(* CODESYS project Screen_1.xml

Project tree, tasks and I/O mapping:
  visualisation Screen_1
*)

// /Screen_1
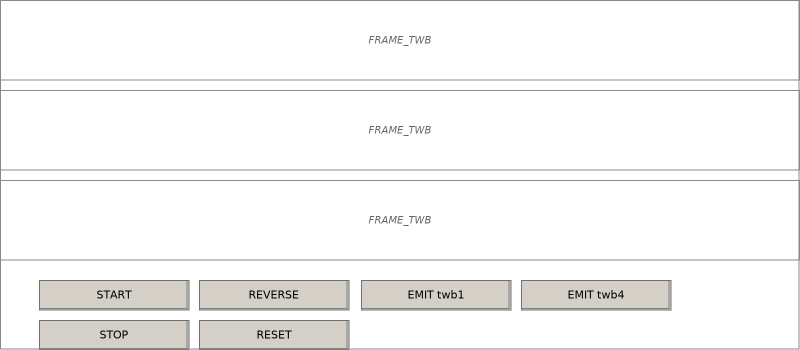
VISUALIZATION Screen_1  // 800x350
    Frame (0,0 800x80)
        shows FRAME_TWB(conveyor := ZONE_HMI.arConveyors[1])
    Frame (0,90 800x80)
        shows FRAME_TWB(conveyor := ZONE_HMI.arConveyors[2])
    Frame (0,180 800x80)
        shows FRAME_TWB(conveyor := ZONE_HMI.arConveyors[3])
    Button (39,280 150x30), "START"
        OnMouseClick: execute { ZONE_HMI.xStart := TRUE; }
    Button (199,280 150x30), "REVERSE"
        OnMouseClick:  ToggleVariable=ZONE_HMI.xReverse
    Button (361,280 150x30), "EMIT twb1"
        OnMouseClick:  ToggleVariable=ZONE_HMI.xEmitt1
    Button (521,280 150x30), "EMIT twb4"
        OnMouseClick:  ToggleVariable=ZONE_HMI.xEmitt2
    Button (39,320 150x30), "STOP"
        OnMouseClick: execute { ZONE_HMI.xStop := TRUE; }
    Button (199,320 150x30), "RESET"
        OnMouseClick: execute { ZONE_HMI.xReset := TRUE; }
END_VISUALIZATION
